(* IEC 61131-3 sources: Sliding-door-with-sensors/Sliding-door_with_sensors/build, 2 files *)

(* ---- plc.st ---- *)
TYPE
  LOGLEVEL : (CRITICAL, WARNING, INFO, DEBUG) := INFO;
END_TYPE

FUNCTION_BLOCK LOGGER
  VAR_INPUT
    TRIG : BOOL;
    MSG : STRING;
    LEVEL : LOGLEVEL := INFO;
  END_VAR
  VAR
    TRIG0 : BOOL;
  END_VAR

  IF TRIG AND NOT TRIG0 THEN
  {{
   LogMessage(GetFbVar(LEVEL),(char*)GetFbVar(MSG, .body),GetFbVar(MSG, .len));
  }}
  END_IF;
  TRIG0:=TRIG;
END_FUNCTION_BLOCK

FUNCTION_BLOCK python_eval
  VAR_INPUT
    TRIG : BOOL;
    CODE : STRING;
  END_VAR
  VAR_OUTPUT
    ACK : BOOL;
    RESULT : STRING;
  END_VAR
  VAR
    STATE : DWORD;
    BUFFER : STRING;
    PREBUFFER : STRING;
    TRIGM1 : BOOL;
    TRIGGED : BOOL;
  END_VAR

  {extern void __PythonEvalFB(int, PYTHON_EVAL*);__PythonEvalFB(0, data__);}
END_FUNCTION_BLOCK

FUNCTION_BLOCK python_poll
  VAR_INPUT
    TRIG : BOOL;
    CODE : STRING;
  END_VAR
  VAR_OUTPUT
    ACK : BOOL;
    RESULT : STRING;
  END_VAR
  VAR
    STATE : DWORD;
    BUFFER : STRING;
    PREBUFFER : STRING;
    TRIGM1 : BOOL;
    TRIGGED : BOOL;
  END_VAR

  {extern void __PythonEvalFB(int, PYTHON_EVAL*);__PythonEvalFB(1,(PYTHON_EVAL*)(void*)data__);}
END_FUNCTION_BLOCK

FUNCTION_BLOCK python_gear
  VAR_INPUT
    N : UINT;
    TRIG : BOOL;
    CODE : STRING;
  END_VAR
  VAR_OUTPUT
    ACK : BOOL;
    RESULT : STRING;
  END_VAR
  VAR
    py_eval : python_eval;
    COUNTER : UINT;
    _TMP_ADD10_OUT : UINT;
    _TMP_EQ13_OUT : BOOL;
    _TMP_SEL15_OUT : UINT;
    _TMP_AND7_OUT : BOOL;
  END_VAR

  _TMP_ADD10_OUT := ADD(COUNTER, 1);
  _TMP_EQ13_OUT := EQ(N, _TMP_ADD10_OUT);
  _TMP_SEL15_OUT := SEL(_TMP_EQ13_OUT, _TMP_ADD10_OUT, 0);
  COUNTER := _TMP_SEL15_OUT;
  _TMP_AND7_OUT := AND(_TMP_EQ13_OUT, TRIG);
  py_eval(TRIG := _TMP_AND7_OUT, CODE := CODE);
  ACK := py_eval.ACK;
  RESULT := py_eval.RESULT;
END_FUNCTION_BLOCK

PROGRAM Sliding_door_with_sensors
  VAR_INPUT RETAIN
    X0 : BOOL := 0;
  END_VAR
  VAR_INPUT
    X1 : BOOL;
    X2 : BOOL;
  END_VAR
  VAR_OUTPUT
    Y0 : BOOL;
    Y1 : BOOL;
  END_VAR
  VAR_IN_OUT
    Zs : BOOL;
  END_VAR
  VAR
    RS0 : RS;
    TON0 : TON;
    SR1 : SR;
    _TMP_NOT19_OUT : BOOL;
    _TMP_AND18_OUT : BOOL;
    _TMP_AND7_OUT : BOOL;
    _TMP_OR9_OUT : BOOL;
  END_VAR

  RS0(S := X0, R1 := X2);
  Y0 := RS0.Q1;
  _TMP_NOT19_OUT := NOT(X0);
  _TMP_AND18_OUT := AND(_TMP_NOT19_OUT, X2);
  TON0(IN := _TMP_AND18_OUT, PT := T#2m);
  Zs := TON0.Q;
  _TMP_AND7_OUT := AND(_TMP_NOT19_OUT, Zs);
  _TMP_OR9_OUT := OR(X0, X1);
  SR1(S1 := _TMP_AND7_OUT, R := _TMP_OR9_OUT);
  Y1 := SR1.Q1;
END_PROGRAM

CONFIGURATION Config0

  RESOURCE Res0 ON PLC
    TASK task0(INTERVAL := T#20ms,PRIORITY := 0);
    PROGRAM instance0 WITH task0 : Sliding_door_with_sensors;
  END_RESOURCE
END_CONFIGURATION

(* ---- generated_plc.st ---- *)
PROGRAM Sliding_door_with_sensors
  VAR_INPUT RETAIN
    X0 : BOOL := 0;
  END_VAR
  VAR_INPUT
    X1 : BOOL;
    X2 : BOOL;
  END_VAR
  VAR_OUTPUT
    Y0 : BOOL;
    Y1 : BOOL;
  END_VAR
  VAR_IN_OUT
    Zs : BOOL;
  END_VAR
  VAR
    RS0 : RS;
    TON0 : TON;
    SR1 : SR;
    _TMP_NOT19_OUT : BOOL;
    _TMP_AND18_OUT : BOOL;
    _TMP_AND7_OUT : BOOL;
    _TMP_OR9_OUT : BOOL;
  END_VAR

  RS0(S := X0, R1 := X2);
  Y0 := RS0.Q1;
  _TMP_NOT19_OUT := NOT(X0);
  _TMP_AND18_OUT := AND(_TMP_NOT19_OUT, X2);
  TON0(IN := _TMP_AND18_OUT, PT := T#2m);
  Zs := TON0.Q;
  _TMP_AND7_OUT := AND(_TMP_NOT19_OUT, Zs);
  _TMP_OR9_OUT := OR(X0, X1);
  SR1(S1 := _TMP_AND7_OUT, R := _TMP_OR9_OUT);
  Y1 := SR1.Q1;
END_PROGRAM

CONFIGURATION Config0

  RESOURCE Res0 ON PLC
    TASK task0(INTERVAL := T#20ms,PRIORITY := 0);
    PROGRAM instance0 WITH task0 : Sliding_door_with_sensors;
  END_RESOURCE
END_CONFIGURATION
